TYPE E_SlaveArmState :
(
	SlaveArmState_Error := 1,
	SlaveArmState_Init :=2,
	SlaveArmState_SelfCheck :=3,
	SlaveArmState_Standby :=4,
	SlaveArmState_MountPanel:=5,
	SlaveArmState_PanelReady :=6,
	SlaveArmState_MountInstru :=7,
	SlaveArmState_InstruReady :=8,
	SlaveArmState_MasterSlave :=9,
	SlaveArmState_ScopeReady :=10,
	SlaveArmState_EndoScope :=11,
	SlaveArmState_Adjust :=12,
	SlaveArmState_Package :=13,
	SlaveArmState_Cart := 14,
	SlaveArmState_GravityCali := 15,
	SlaveArmState_Test := 16,
	SlaveArmState_InstruRetract :=17,
	SlaveArmState_InstruInvasion :=18,
	SlaveArmState_Disable := 19,
	SlaveArmState_InstruCali := 20,
	SlaveArmState_ScopeToggle :=21,
	SlaveArmState_Performance:=22,
	SlaveArmState_Stop :=23,
	SlaveArmState_InstruAutoTest :=24,
	SlaveArmState_InstruManualTest :=25,
	SlaveArmState_InstruVerify :=26,
	SlaveArmState_MotorGoHome:= 27,
	SlaveArmState_PowerBoxCalibration:= 28,
	SlaveArmState_EndoscopeTest:= 29,
	SlaveArmState_FrictionTest:= 30,
	
	SlaveArmState_Jnt5Rotate:=31,
	SlaveArmState_totalNum :=SlaveArmState_Jnt5Rotate
);
END_TYPE

(* stored: Version 1.1.0.1, ProductVersion 3.1.4024.11
   DUT E_SlaveArmState: Id {1989848d-a357-4300-a3bc-ded8b39d8e17} *)
